# EPICS substitutions: l2MpsAsynApp/Db/mps_blen.substitutions
### Threshold information ###
file "RegRO.template" { pattern
{ R,                DESC,                               PARAM,              ADDR        }
{ L_THR_CH,         "Bay $(BAY) Threshold channel",     BLEN_THRNUM_0,      "$(BAY)"    }
{ L_THR_CNT,        "Bay $(BAY) Threshold count",       BLEN_THRCNT_0,      "$(BAY)"    }
{ L_THR_BYTEMAP,    "Bay $(BAY) Threshold byte map",    BLEN_BYTEMAP_0,     "$(BAY)"    }
{ L_LATCHED_RAW,    "Bay $(BAY) Latched Value",         BLEN_TRIP_VALUER_0, "$(BAY)"    }
}

file "RegROFloat.template" { pattern
{ R,                DESC,                                      EGU,     PARAM,              ADDR        }
{ L_LATCHED,       "Bay $(BAY) Latched Value",                 "",      BLEN_TRIP_VALUE_0,  "$(BAY)"    }
}

file "RegRO64.template" { pattern
{ R,                DESC,                                          PARAM,             ADDR        }
{ L_LATCHED_PID,    "Bay $(BAY) Latched PID",                      BLEN_TRIP_PID_0,   "$(BAY)"    }
}

### Tables enable PVs ###
file "Reg1BitRW.template" { pattern
{ R,                DESC,                               PARAM,              ADDR,       ZNAM,           ONAM        }
{ L_IDL_EN,         "Bay $(BAY) IDLE table enabled",    BLEN_IDLEEN_0,      "$(BAY)",   "Disabled",     "Enabled"   }
}

file "Reg1BitRO.template" { pattern
{ R,                DESC,                               PARAM,              ADDR,       ZNAM,           ONAM        }
{ L_ALT_EN,         "Bay $(BAY) ALT table enabled",     BLEN_ALTEN_0,       "$(BAY)",   "Disabled",     "Enabled"   }
{ L_LC1_EN,         "Bay $(BAY) LCLS1 table enabled",   BLEN_LCLS1EN_0,     "$(BAY)",   "Disabled",     "Enabled"   }
}

### Threshold PVs ###
file "thr.template" { pattern
{ R,                DESC,                                   APP,        CH,     TABLE,  THR,    }
{ L_T0_LC1,         "BLEN, Bay $(BAY), LCLS1, Threshold",   "BLEN",     "0",    "0",    "0",    }

{ L_T0_IDL,         "BLEN, Bay $(BAY), IDLE, Threshold",    "BLEN",     "0",    "1",    "0",    }

{ L_T0,             "BLEN, Bay $(BAY), STD, Threshold 0",   "BLEN",     "0",    "2",    "0",    }
{ L_T1,             "BLEN, Bay $(BAY), STD, Threshold 1",   "BLEN",     "0",    "2",    "1",    }
{ L_T2,             "BLEN, Bay $(BAY), STD, Threshold 2",   "BLEN",     "0",    "2",    "2",    }
{ L_T3,             "BLEN, Bay $(BAY), STD, Threshold 3",   "BLEN",     "0",    "2",    "3",    }
{ L_T4,             "BLEN, Bay $(BAY), STD, Threshold 4",   "BLEN",     "0",    "2",    "4",    }
{ L_T5,             "BLEN, Bay $(BAY), STD, Threshold 5",   "BLEN",     "0",    "2",    "5",    }
{ L_T6,             "BLEN, Bay $(BAY), STD, Threshold 6",   "BLEN",     "0",    "2",    "6",    }
{ L_T7,             "BLEN, Bay $(BAY), STD, Threshold 7",   "BLEN",     "0",    "2",    "7",    }

{ L_T0_ALT,         "BLEN, Bay $(BAY), ALT, Threshold 0",   "BLEN",     "0",    "3",    "0",    }
{ L_T1_ALT,         "BLEN, Bay $(BAY), ALT, Threshold 1",   "BLEN",     "0",    "3",    "1",    }
{ L_T2_ALT,         "BLEN, Bay $(BAY), ALT, Threshold 2",   "BLEN",     "0",    "3",    "2",    }
{ L_T3_ALT,         "BLEN, Bay $(BAY), ALT, Threshold 3",   "BLEN",     "0",    "3",    "3",    }
{ L_T4_ALT,         "BLEN, Bay $(BAY), ALT, Threshold 4",   "BLEN",     "0",    "3",    "4",    }
{ L_T5_ALT,         "BLEN, Bay $(BAY), ALT, Threshold 5",   "BLEN",     "0",    "3",    "5",    }
{ L_T6_ALT,         "BLEN, Bay $(BAY), ALT, Threshold 6",   "BLEN",     "0",    "3",    "6",    }
{ L_T7_ALT,         "BLEN, Bay $(BAY), ALT, Threshold 7",   "BLEN",     "0",    "3",    "7",    }
}

### Scale PVs ###
file "scale.template" { pattern
{ R,        DESC,                           APP,        EGU,    PREC,   CH,     SCALE_SLOPE_PV,     SCALE_OFFSET_PV,    SCAN        }
{ L,        "Bay $(BAY) Scale factor",      "BLEN",     "",     "4",    "0",    "$(P):L_FWSLO",     "$(P):L_FWOFF",     "1 second"  }
}

file "name.template" { pattern
{ R,   PARAM,         ADDR    }
{ L,   "BLEN_NAME_0", "$(BAY)"}
}
